TYPE TcoRoboticsBasicCoordinates : 
STRUCT
    {attribute  addProperty Name "<#Coordinate X#>"}
    X : REAL;
    {attribute  addProperty Name "<#Coordinate Y#>"}
    Y : REAL;
    {attribute  addProperty Name "<#Coordinate Z#>"}
    Z : REAL;
END_STRUCT
END_TYPE

(* stored: Version 1.1.0.1, ProductVersion 3.1.4024.12
   DUT TcoRoboticsBasicCoordinates: Id {78657219-302a-02f5-3d19-b2c89c9dc730} *)
